// TwinCAT 3 PLC project PLC1
// ProgramVersion: 3.1.4020.4
// libraries:
//   Tc2_Standard, * (Beckhoff Automation GmbH)
//   Tc2_System, * (Beckhoff Automation GmbH)
//   Tc2_TcpIp, * (Beckhoff Automation GmbH)
//   Tc2_Utilities, * (Beckhoff Automation GmbH)
//   Tc3_Module, * (Beckhoff Automation GmbH)
// project tree:
//   HTTP/DUTs/ E_HTTP_Request_Type.TcDUT, ST_HTTP_Connection_Parameters.TcDUT, ST_HTTP_Parameter.TcDUT, ST_HTTP_Request.TcDUT, ST_HTTP_Response.TcDUT
//   HTTP/ FB_Http_Client.TcPOU
//   HTTP/GVLs/ GVL_HTTP.TcGVL
//   HTTP/Helper POUs/ FB_BinaryWriter.TcPOU, FB_GetHttpConnectionParams.TcPOU, F_BuildHttpGetRequest.TcPOU, F_BuildHttpPostRequest.TcPOU, F_MultiConcat12.TcPOU, F_MultiConcat6.TcPOU, F_ParseHttpResponse.TcPOU, F_ParseHttpUrl.TcPOU
//   HTTP/InfluxDb/ FB_Http_Client_Influx.TcPOU, F_BuildHttpPostRequest_InfluxDb.TcPOU
//   / PlcTask.TcTTO
//   POUs/ MAIN.TcPOU
// real-time tasks:
//   TASK PlcTask: cycle T#10ms, priority 20, ADS port 350

CONFIGURATION PLC1
    RESOURCE PLC ON TwinCAT3
        TASK PlcTask(INTERVAL := T#10ms, PRIORITY := 20);
        PROGRAM MAIN WITH PlcTask : MAIN;
    END_RESOURCE
END_CONFIGURATION

// ---- HTTP/DUTs/E_HTTP_Request_Type.TcDUT
TYPE E_HTTP_Request_Type :
(
	E_HTTP_Request_Type_GET := 0,
	E_HTTP_Request_Type_POST := 1
);
END_TYPE

// ---- HTTP/DUTs/ST_HTTP_Connection_Parameters.TcDUT
TYPE ST_HTTP_Connection_Parameters :
STRUCT
	bIsValid		: BOOL;
	sIpv4Address	: STRING;
	udPort			: UDINT;
	sHostName		: STRING;
	sRequestURI 	: STRING;
END_STRUCT
END_TYPE

// ---- HTTP/DUTs/ST_HTTP_Parameter.TcDUT
TYPE ST_HTTP_Parameter :
STRUCT
	sName	: STRING;
	sValue	: STRING;
END_STRUCT
END_TYPE

// ---- HTTP/DUTs/ST_HTTP_Request.TcDUT
TYPE ST_HTTP_Request :
STRUCT
	eHttpRequestType	: E_HTTP_Request_Type;
	arrParameters 		: ARRAY [0..HTTP_PARAMETERS_ARRAY_SIZE] OF ST_HTTP_Parameter;
END_STRUCT
END_TYPE

// ---- HTTP/DUTs/ST_HTTP_Response.TcDUT
TYPE ST_HTTP_Response :
STRUCT
	arrHeaders	: ARRAY [0..HTTP_RESPONSE_HEADER_ARRAY_SIZE] OF STRING;
	sContent	: STRING(255);
END_STRUCT
END_TYPE

// ---- HTTP/GVLs/GVL_HTTP.TcGVL
VAR_GLOBAL CONSTANT
	HTTP_SEND_DATA_ARRAY_SIZE 		: UDINT := 49999; 
	HTTP_RECEIVE_DATA_ARRAY_SIZE 	: UDINT := 9999; 
	HTTP_PARAMETERS_ARRAY_SIZE		: UDINT := 499;
	HTTP_RESPONSE_HEADER_ARRAY_SIZE	: UDINT := 20; 
END_VAR

// ---- POUs/MAIN.TcPOU
PROGRAM MAIN
VAR
	fbHttp_ClientPost	: FB_Http_Client;
	stHttpReqPost		: ST_HTTP_Request; 
	stHttpResponsePost	: ST_HTTP_Response;
	sResponsePost		: STRING(255);
	T1_TON				: TON;
	
	fbHttp_ClientGet	: FB_Http_Client;
	stHttpReqGet		: ST_HTTP_Request; 
	stHttpResponseGet	: ST_HTTP_Response;
	T2_TON				: TON;
	sResponseGet		: STRING(255);
	udCounter			: UDINT;
END_VAR

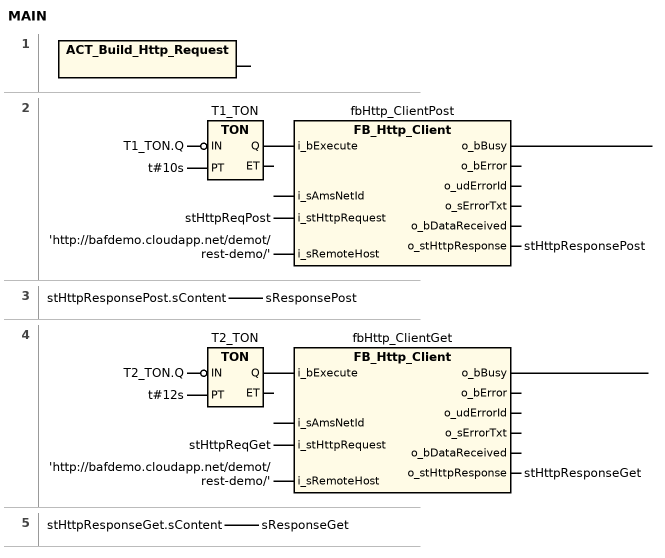
// NETWORK 1
ACT_Build_Http_Request();

// NETWORK 2
T1_TON(IN := NOT T1_TON.Q, PT := t#10s); // TON
fbHttp_ClientPost(
    i_bExecute := T1_TON.Q,
    i_stHttpRequest := stHttpReqPost,
    i_sRemoteHost := 'http://bafdemo.cloudapp.net/demot/rest-demo/',
    o_stHttpResponse => stHttpResponsePost); // FB_Http_Client

// NETWORK 3
sResponsePost := stHttpResponsePost.sContent;

// NETWORK 4
T2_TON(IN := NOT T2_TON.Q, PT := t#12s); // TON
fbHttp_ClientGet(
    i_bExecute := T2_TON.Q,
    i_stHttpRequest := stHttpReqGet,
    i_sRemoteHost := 'http://bafdemo.cloudapp.net/demot/rest-demo/',
    o_stHttpResponse => stHttpResponseGet); // FB_Http_Client

// NETWORK 5
sResponseGet := stHttpResponseGet.sContent;

ACTION ACT_Build_Http_Request:

(****  HTTP POST Example ********************************************************************************)

stHttpReqPost.eHttpRequestType 			:= E_HTTP_Request_Type.E_HTTP_Request_Type_POST;

stHttpReqPost.arrParameters[0].sName	:= 'passwd';
stHttpReqPost.arrParameters[0].sValue	:= 'TwoCats';

stHttpReqPost.arrParameters[1].sName	:= 'counter';
stHttpReqPost.arrParameters[1].sValue	:= UDINT_TO_STRING(udCounter);  udCounter := udCounter + 1;

stHttpReqPost.arrParameters[2].sName	:= 'cyclecount';
stHttpReqPost.arrParameters[2].sValue	:= UDINT_TO_STRING(_TaskInfo[1].CycleCount);

(*******************************************************************************************************)

(****  HTTP GET Example ********************************************************************************)

stHttpReqGet.eHttpRequestType 			:= E_HTTP_Request_Type.E_HTTP_Request_Type_GET;

stHttpReqGet.arrParameters[0].sName		:= 'passwd';
stHttpReqGet.arrParameters[0].sValue	:= 'TwoCats';

stHttpReqGet.arrParameters[1].sName		:= 'parameters';
stHttpReqGet.arrParameters[1].sValue	:= '1';

(*******************************************************************************************************)
END_ACTION

END_PROGRAM

// ---- HTTP/FB_Http_Client.TcPOU
FUNCTION_BLOCK FB_Http_Client
VAR_INPUT
	i_bExecute 			: BOOL;
	i_sAmsNetId			: STRING;
	i_stHttpRequest 	: ST_HTTP_Request;
	i_sRemoteHost		: STRING(255);
END_VAR
VAR_OUTPUT	
	o_bBusy				: BOOL;
	o_bError			: BOOL;
	o_udErrorId			: UDINT;
	o_sErrorTxt			: STRING;
	o_bDataReceived		: BOOL;	
	o_stHttpResponse	: ST_HTTP_Response;
END_VAR
VAR
	fbGetHttpConnectionParams: FB_GetHttpConnectionParams;
	fbSocketConnect		: FB_SocketConnect;
	fbSocketSend		: FB_SocketSend;
	fbSocketReceive		: FB_SocketReceive;
	fbSocketClose		: FB_SocketClose;
	bGetHttpConnectionParams: BOOL;
	bSocketConnect		: BOOL;
	bSocketSend			: BOOL;
	bSocketReceive		: BOOL;
	bSocketClose		: BOOL;
	nState				: INT := 10;
	hSocket				: T_HSOCKET;
	udBytesToSend		: UDINT;
	arrBytesToSend		: ARRAY[0..HTTP_SEND_DATA_ARRAY_SIZE] OF BYTE;
	tTimeOut			: TIME := T#10S;
	arrReceivedBytes	: ARRAY[0..HTTP_RECEIVE_DATA_ARRAY_SIZE] OF BYTE;
	bHttpConnParamsParamsParsed : BOOL;
	stHttpConnectionParams : ST_HTTP_Connection_Parameters;
	udReceivedBytes		: UDINT;
	Delay_TON			: TON;
END_VAR



CASE nState OF

10: (* Initial state *)
	nState := 20;
	
20:	(* Waiting for start *)

	IF i_bExecute THEN
		
		MEMSET(ADR(arrReceivedBytes), 0, SIZEOF(arrReceivedBytes));
		o_bDataReceived := FALSE;
		udReceivedBytes := 0;
		o_udErrorId		:= 0;
		o_bError 		:= FALSE;
		o_sErrorTxt 	:= '';
		o_bBusy 		:= TRUE;
		
		IF NOT bHttpConnParamsParamsParsed THEN
			bGetHttpConnectionParams := TRUE;
			nState := 25;
		ELSE
			bSocketConnect 	:= TRUE;
			nState 			:= 30;
		END_IF
		
	END_IF

25:	(* Waiting for addr resolved *)


	IF fbGetHttpConnectionParams.o_bError THEN
		o_udErrorId := fbGetHttpConnectionParams.o_nErrId;
		o_sErrorTxt := 'FB_GetHttpConnectionParams error';
		nState 		:= 100; 
	ELSIF fbGetHttpConnectionParams.o_bReady THEN
		stHttpConnectionParams := fbGetHttpConnectionParams.o_stHttpConnectionParams;
		bHttpConnParamsParamsParsed := TRUE;
		bSocketConnect 	:= TRUE;
		nState 			:= 30;
	END_IF	

30:	(* Waiting for connect *)

	IF fbSocketConnect.bError THEN
		o_udErrorId := fbSocketConnect.nErrId;
		o_sErrorTxt := 'FB_SocketConnect error';
		nState 		:= 100; 
	ELSIF NOT fbSocketConnect.bBusy THEN
		
		CASE i_stHttpRequest.eHttpRequestType OF 
			
			E_HTTP_Request_Type_GET:			
					udBytesToSend 	:= F_BuildHttpGetRequest(ADR(i_stHttpRequest), stHttpConnectionParams, arrBytesToSend);
							
			E_HTTP_Request_Type_POST:			
					udBytesToSend 	:= F_BuildHttpPostRequest(ADR(i_stHttpRequest), stHttpConnectionParams, arrBytesToSend);
							
		END_CASE

		bSocketSend		:= TRUE;
		nState 			:= 40; 		
	END_IF

40:	(* Waiting for send *) 

	IF fbSocketSend.bError THEN
		o_udErrorId := fbSocketSend.nErrId;
		o_sErrorTxt := 'FB_SocketSend error';
		nState 		:= 100; 
	ELSIF NOT fbSocketSend.bBusy THEN
		bSocketReceive	:= TRUE;
		nState 			:= 50; 		
	END_IF
	
50:	(* Waiting for receive *)

	// Timeout
	Delay_TON(IN := TRUE, PT := T#1500MS);
	
	IF fbSocketReceive.bError THEN
		Delay_TON(IN := FALSE);
		o_udErrorId := fbSocketReceive.nErrId;
		o_sErrorTxt := 'FB_SocketReceive error';
		nState 		:= 100; 
	ELSIF NOT fbSocketReceive.bBusy THEN
		IF fbSocketReceive.nRecBytes > 0 THEN
			Delay_TON(IN := FALSE);
			o_bDataReceived := TRUE;
			udReceivedBytes := fbSocketReceive.nRecBytes;
			o_stHttpResponse:= F_ParseHttpResponse(i_udNumOfBytes := udReceivedBytes, io_arrReceivedBytes:= arrReceivedBytes);
			bSocketClose	:= TRUE;
			nState 			:= 60;
		ELSIF Delay_TON.Q THEN
			Delay_TON(IN := FALSE);
			bSocketClose	:= TRUE;
			nState 			:= 60;
		ELSE
			bSocketReceive	:= TRUE;
		END_IF
	END_IF

60:	(* Waiting for close *)

	IF fbSocketClose.bError THEN
		o_udErrorId := fbSocketClose.nErrId;
		o_sErrorTxt := 'FB_SocketReceive error';
		nState 		:= 100; 
	ELSIF NOT fbSocketClose.bBusy THEN
		nState 	:= 10; 		
		o_bBusy := FALSE;
	END_IF

100:	(* Error *)

	o_bBusy  := FALSE;
	o_bError := TRUE;
	IF NOT i_bExecute THEN
		nState := 10;
	END_IF

END_CASE

ACT_FB_Calls();

bGetHttpConnectionParams := FALSE;
bSocketConnect 	:= FALSE;
bSocketSend 	:= FALSE;
bSocketReceive 	:= FALSE;
bSocketClose 	:= FALSE;

ACTION ACT_FB_Calls:
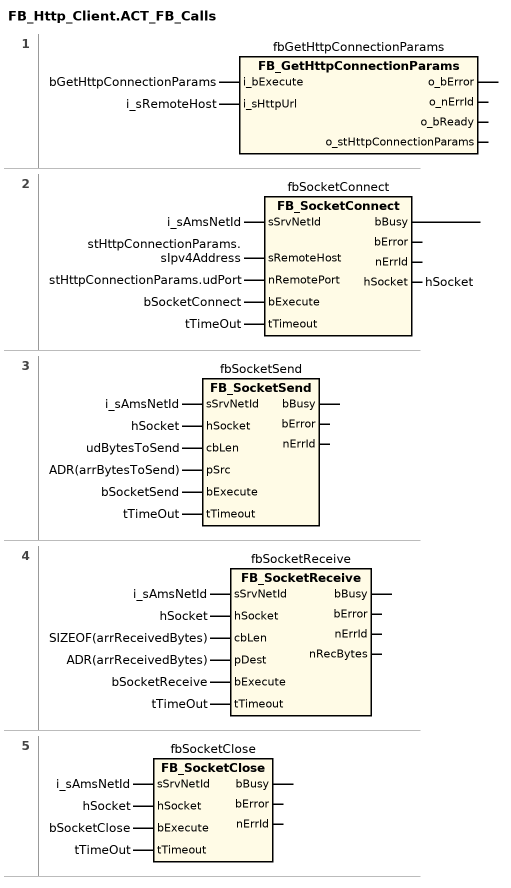
// NETWORK 1
fbGetHttpConnectionParams(i_bExecute := bGetHttpConnectionParams, i_sHttpUrl := i_sRemoteHost); // FB_GetHttpConnectionParams

// NETWORK 2
fbSocketConnect(
    sSrvNetId := i_sAmsNetId,
    sRemoteHost := stHttpConnectionParams.sIpv4Address,
    nRemotePort := stHttpConnectionParams.udPort,
    bExecute := bSocketConnect,
    tTimeout := tTimeOut,
    hSocket => hSocket); // FB_SocketConnect

// NETWORK 3
fbSocketSend(
    sSrvNetId := i_sAmsNetId,
    hSocket := hSocket,
    cbLen := udBytesToSend,
    pSrc := ADR(arrBytesToSend),
    bExecute := bSocketSend,
    tTimeout := tTimeOut); // FB_SocketSend

// NETWORK 4
fbSocketReceive(
    sSrvNetId := i_sAmsNetId,
    hSocket := hSocket,
    cbLen := SIZEOF(arrReceivedBytes),
    pDest := ADR(arrReceivedBytes),
    bExecute := bSocketReceive,
    tTimeout := tTimeOut); // FB_SocketReceive

// NETWORK 5
fbSocketClose(sSrvNetId := i_sAmsNetId, hSocket := hSocket, bExecute := bSocketClose, tTimeout := tTimeOut); // FB_SocketClose
END_ACTION

END_FUNCTION_BLOCK

// ---- HTTP/Helper POUs/FB_GetHttpConnectionParams.TcPOU
FUNCTION_BLOCK FB_GetHttpConnectionParams
VAR_INPUT
	i_bExecute	: BOOL;
	i_sHttpUrl	: T_MaxString;
END_VAR
VAR_OUTPUT
	o_bError	: BOOL;
	o_nErrId	: UDINT;
	o_bReady	: BOOL;
	o_stHttpConnectionParams : ST_HTTP_Connection_Parameters;
END_VAR
VAR
	fbGetHostAddrByName		: FB_GetHostAddrByName;
	stHttpConnectionParams 	: ST_HTTP_Connection_Parameters;
	execute_R_TRIG			: R_TRIG;
	getHostAddrBusy_F_TRIG	: F_TRIG;
	bExecute				: BOOL;
	bUrlValid: BOOL;
	nState: INT := 10;
END_VAR



CASE nState OF
	
10: (* init *)
	nState := 20;
	
20:	(* Waiting for start *)
	
	IF i_bExecute THEN
		(* Reset *)
		o_bReady := FALSE;
		o_bError := FALSE;
		o_nErrId := 0;
		MEMSET(ADR(o_stHttpConnectionParams), 0, SIZEOF(o_stHttpConnectionParams));
		
		IF F_ParseHttpUrl(i_sHttpUrl, stHttpConnectionParams) THEN
			IF stHttpConnectionParams.sHostName <> 'localhost' THEN

				nState := 30;
			ELSE
				stHttpConnectionParams.sIpv4Address := '127.0.0.1';	
				o_stHttpConnectionParams := stHttpConnectionParams;
				o_bReady := TRUE;
				nState := 20;			
			END_IF
		ELSE 
			o_bError := TRUE;
		END_IF
	END_IF

30:	(* Waiting for ready *)

	fbGetHostAddrByName(
		sHostName	:= stHttpConnectionParams.sHostName,
		bExecute 	:= TRUE,
		tTimeout 	:= T#10S
	);
	
	IF fbGetHostAddrByName.bError THEN
		fbGetHostAddrByName(bExecute := FALSE);
		o_bError := TRUE;
		o_nErrId := fbGetHostAddrByName.nErrID;
		nState := 100;
	ELSIF NOT fbGetHostAddrByName.bBusy THEN
		fbGetHostAddrByName(bExecute := FALSE);
		stHttpConnectionParams.sIpv4Address := fbGetHostAddrByName.sAddr;
		o_stHttpConnectionParams := stHttpConnectionParams;
		o_bReady := TRUE;
		nState := 20;
	END_IF
	
100: (* Error state*)

	IF NOT i_bExecute THEN
		nState := 10;
	END_IF

END_CASE

END_FUNCTION_BLOCK

// ---- HTTP/Helper POUs/F_ParseHttpUrl.TcPOU
FUNCTION F_ParseHttpUrl : BOOL
VAR_INPUT
	i_sUrl :T_MaxString;
END_VAR
VAR_IN_OUT 
	io_stConnectionParameters : ST_HTTP_Connection_Parameters;
END_VAR
VAR
	sUrl : T_MaxString;
	stConnectionParameters : ST_HTTP_Connection_Parameters;
	nPos: INT;
	nPosPort: INT;
END_VAR

sUrl := i_sUrl;

//the shortest form http://a.fi ==> 11 characters
IF LEN(sUrl) < 11 THEN
	F_ParseHttpUrl := FALSE;
	RETURN;
END_IF

// Parse the protocol
IF LEFT(sUrl, 5) = 'https' THEN
	// HTTPS is not supported
	F_ParseHttpUrl := FALSE;
	RETURN;
ELSIF LEFT(sUrl, 4) = 'http' THEN
	stConnectionParameters.udPort := 80;
	sUrl := RIGHT(sUrl, LEN(sUrl) - 4);
ELSE
	F_ParseHttpUrl := FALSE;
	RETURN;
END_IF

//Remove '://'
IF LEFT(sUrl, 3) = '://' THEN
	sUrl := RIGHT(sUrl, LEN(sUrl) - 3);
	// There is only domain + request uri left, minimun 4 characters (a.fi)
	IF LEN(sUrl) < 4 THEN 
		F_ParseHttpUrl := FALSE;
		RETURN;
	END_IF
ELSE
	F_ParseHttpUrl := FALSE;
	RETURN;
END_IF

// We have domain [+ port [+ request uri]] left
nPos := FIND(sUrl, '/');
nPosPort := FIND(sUrl, ':');

IF nPos = 0 THEN
	IF nPosPort > 0 THEN
		stConnectionParameters.sHostName := LEFT(sUrl, nPosPort-1);
		sUrl := RIGHT(sUrl, LEN(sUrl) - nPosPort);		
	ELSE
		stConnectionParameters.sHostName := sUrl;
	END_IF
	stConnectionParameters.sRequestURI := '/';
	io_stConnectionParameters := stConnectionParameters;
	F_ParseHttpUrl := TRUE;
ELSE
	IF nPosPort > 0 THEN
		stConnectionParameters.sHostName := LEFT(sUrl, nPosPort-1);
		sUrl := RIGHT(sUrl, LEN(sUrl) - nPosPort);		
		nPos := FIND(sUrl, '/');
		stConnectionParameters.udPort := STRING_TO_UDINT(LEFT(sUrl, nPos-1));
		sUrl := RIGHT(sUrl, LEN(sUrl) - nPos + 1);	
	ELSE
		stConnectionParameters.sHostName := LEFT(sUrl, nPos-1);
		sUrl := RIGHT(sUrl, LEN(sUrl) - nPos+1);
	END_IF	
	stConnectionParameters.sRequestURI := sUrl;
	io_stConnectionParameters := stConnectionParameters;
	F_ParseHttpUrl := TRUE;
END_IF

END_FUNCTION

// ---- HTTP/Helper POUs/F_BuildHttpGetRequest.TcPOU
FUNCTION F_BuildHttpGetRequest : UDINT
VAR_INPUT
	i_pHttpRequest 		: POINTER TO ST_HTTP_Request;
	i_stHttpConnParams	: ST_HTTP_Connection_Parameters;
END_VAR
VAR_IN_OUT
	io_arrBytesToSend	: ARRAY[0..HTTP_SEND_DATA_ARRAY_SIZE] OF BYTE;
END_VAR
VAR
	sData				: T_MaxString;
	i					: INT;
	nContentLength		: DINT;
	fbBinaryWriter		: FB_BinaryWriter;
	sRequestString		: STRING(255);
END_VAR


fbBinaryWriter.Init(ADR(io_arrBytesToSend), SIZEOF(io_arrBytesToSend));
MEMSET(ADR(io_arrBytesToSend), 0, SIZEOF(io_arrBytesToSend));

fbBinaryWriter.WriteString('GET ');
fbBinaryWriter.WriteString(i_stHttpConnParams.sRequestURI);

// Write the GET request into request uri
FOR i := 0 TO UDINT_TO_INT(HTTP_PARAMETERS_ARRAY_SIZE) DO 
	IF LEN(i_pHttpRequest^.arrParameters[i].sName) > 0 THEN
		IF i = 0 THEN fbBinaryWriter.WriteString('?'); END_IF
		IF i > 0 THEN fbBinaryWriter.WriteString('&'); END_IF
		fbBinaryWriter.WriteString(i_pHttpRequest^.arrParameters[i].sName);
		fbBinaryWriter.WriteString('=');
		fbBinaryWriter.WriteString(i_pHttpRequest^.arrParameters[i].sValue);
	END_IF
END_FOR

fbBinaryWriter.WriteString(' HTTP/1.0$R$N'); // Lets use HTTP 1.0 because responce with "Transfer-Encoding:chunked is much more complex to parse
fbBinaryWriter.WriteString('Host: ');
fbBinaryWriter.WriteString(i_stHttpConnParams.sHostName);
fbBinaryWriter.WriteString(' $R$N');
fbBinaryWriter.WriteString('User-Agent: TwinCAT HttpClient$R$N');

// Calculate the length of data
FOR i := 0 TO UDINT_TO_INT(HTTP_PARAMETERS_ARRAY_SIZE) DO 
	IF LEN(i_pHttpRequest^.arrParameters[i].sName) > 0 THEN
		IF i > 0 THEN nContentLength := nContentLength + 1; END_IF
		nContentLength := nContentLength + LEN(i_pHttpRequest^.arrParameters[i].sName) + LEN(i_pHttpRequest^.arrParameters[i].sValue) + 1;
	END_IF
END_FOR	
fbBinaryWriter.WriteString('$R$N$R$N');
	
sRequestString := fbBinaryWriter.ToString;

F_BuildHttpGetRequest := fbBinaryWriter.Length;

(****** GET Request principle ***********************************************************************

fbBinaryWriter.WriteString('GET /demot/rest-demo/?'param1=1&param2=2&param3=3' HTTP/1.1$R$N');
fbBinaryWriter.WriteString('Host: bafdemo.cloudapp.net $R$N');
fbBinaryWriter.WriteString('User-Agent: TwinCAT 3.1$R$N');
fbBinaryWriter.WriteString('$R$N$R$N');

***************************************************************************************************)

END_FUNCTION

// ---- HTTP/Helper POUs/FB_BinaryWriter.TcPOU
FUNCTION_BLOCK FB_BinaryWriter
VAR_INPUT
	i_pDestAddr		: POINTER TO BYTE;
	i_udDestAddrLen	: UDINT;
END_VAR
VAR_OUTPUT
END_VAR
VAR
	pDestAddr		: POINTER TO BYTE;
	udDestAddrLen	: UDINT;
	udCurrentLen 	: UDINT;
END_VAR

METHOD Init : BOOL
VAR_INPUT
	i_pDestAddr		: POINTER TO BYTE;
	i_udDestAddrLen	: UDINT;
END_VAR
pDestAddr 		:= i_pDestAddr;
udDestAddrLen 	:=i_udDestAddrLen;
udCurrentLen 	:= 0;

(* Reset the stream *)
MEMSET(i_pDestAddr, 0, i_udDestAddrLen);
END_METHOD

PROPERTY Length : udint
GET
Length := udCurrentLen;
END_GET
END_PROPERTY

METHOD SetPosition : BOOL
VAR_INPUT
	i_udPosition : UDINT;
END_VAR
IF i_udPosition <= udDestAddrLen THEN
	udCurrentLen := i_udPosition;
	SetPosition := TRUE;
ELSE
	SetPosition := FALSE;
END_IF
END_METHOD

PROPERTY ToString : STRING(255)
GET
VAR
	s255String : STRING(255);
	length : UDINT;
END_VAR
s255String := '';
length := MIN(udCurrentLen, DINT_TO_UDINT(SIZEOF(s255String)));
MEMCPY(ADR(s255String), pDestAddr, length);
ToString := s255String;
END_GET
END_PROPERTY

METHOD WriteString : BOOL
VAR_INPUT
	i_sStringToAppend : T_MaxString;
END_VAR
VAR
	udStringLen: UDINT;
END_VAR

udStringLen := DINT_TO_UDINT(LEN(i_sStringToAppend));

(* Only write if there's memory free for writing *)
IF udCurrentLen + udStringLen < udDestAddrLen THEN
	MEMCPY(pDestAddr + udCurrentLen, ADR(i_sStringToAppend), udStringLen);
	udCurrentLen := udCurrentLen + udStringLen;
	WriteString := TRUE;
ELSE
	WriteString := FALSE;
END_IF
END_METHOD

END_FUNCTION_BLOCK

// ---- HTTP/Helper POUs/F_BuildHttpPostRequest.TcPOU
FUNCTION F_BuildHttpPostRequest : UDINT
VAR_INPUT
	i_pHttpRequest 		: POINTER TO ST_HTTP_Request;
	i_stHttpConnParams	: ST_HTTP_Connection_Parameters;
END_VAR
VAR_IN_OUT
	io_arrBytesToSend	: ARRAY[0..HTTP_SEND_DATA_ARRAY_SIZE] OF BYTE;
END_VAR
VAR
	sData				: T_MaxString;
	i					: INT;
	nContentLength		: DINT;
	fbBinaryWriter		: FB_BinaryWriter;
	sRequestString		: STRING(255);
END_VAR


fbBinaryWriter.Init(ADR(io_arrBytesToSend), SIZEOF(io_arrBytesToSend));
MEMSET(ADR(io_arrBytesToSend), 0, SIZEOF(io_arrBytesToSend));

fbBinaryWriter.WriteString('POST ');
fbBinaryWriter.WriteString(i_stHttpConnParams.sRequestURI);
fbBinaryWriter.WriteString(' HTTP/1.0$R$N'); // Lets use HTTP 1.0 because responce with "Transfer-Encoding:chunked is much more complex to parse
fbBinaryWriter.WriteString('Host: ');
fbBinaryWriter.WriteString(i_stHttpConnParams.sHostName);
fbBinaryWriter.WriteString(' $R$N');
fbBinaryWriter.WriteString('User-Agent: TwinCAT HttpClient$R$N');
fbBinaryWriter.WriteString('Content-Type: application/x-www-form-urlencoded$R$N');

// Calculate the length of data
FOR i := 0 TO UDINT_TO_INT(HTTP_PARAMETERS_ARRAY_SIZE) DO 
	IF LEN(i_pHttpRequest^.arrParameters[i].sName) > 0 THEN
		IF i > 0 THEN nContentLength := nContentLength + 1; END_IF
		nContentLength := nContentLength + LEN(i_pHttpRequest^.arrParameters[i].sName) + LEN(i_pHttpRequest^.arrParameters[i].sValue) + 1;
	END_IF
END_FOR	

fbBinaryWriter.WriteString(CONCAT('Content-Length: ', DINT_TO_STRING(nContentLength)));


// Http request headers always end to double new line		
fbBinaryWriter.WriteString('$R$N$R$N');

// Write the POST data into request body
FOR i := 0 TO UDINT_TO_INT(HTTP_PARAMETERS_ARRAY_SIZE) DO 
	IF LEN(i_pHttpRequest^.arrParameters[i].sName) > 0 THEN
		IF i > 0 THEN fbBinaryWriter.WriteString('&'); END_IF
		fbBinaryWriter.WriteString(i_pHttpRequest^.arrParameters[i].sName);
		fbBinaryWriter.WriteString('=');
		fbBinaryWriter.WriteString(i_pHttpRequest^.arrParameters[i].sValue);
	END_IF
END_FOR

// Http request body always ends to new line		
fbBinaryWriter.WriteString('$R$N');


sRequestString := fbBinaryWriter.ToString;
F_BuildHttpPostRequest := fbBinaryWriter.Length;

(****** POST Request principle ***********************************************************************

sPostData = 'param1=1&param2=2&param3=3';
fbBinaryWriter.WriteString('POST /demot/rest-demo/ HTTP/1.1$R$N');
fbBinaryWriter.WriteString('Host: bafdemo.cloudapp.net $R$N');
fbBinaryWriter.WriteString('User-Agent: TwinCAT 3.1$R$N');
fbBinaryWriter.WriteString('Content-Type: application/x-www-form-urlencoded$R$N');
fbBinaryWriter.WriteString(CONCAT('Content-Length: ', DINT_TO_STRING(LEN(sPostData))));
fbBinaryWriter.WriteString('$R$N$R$N');
fbBinaryWriter.WriteString(sPostData);
fbBinaryWriter.WriteString('$R$N');

******************************************************************************************************)

END_FUNCTION

// ---- HTTP/Helper POUs/F_ParseHttpResponse.TcPOU
FUNCTION F_ParseHttpResponse : ST_HTTP_Response
VAR_INPUT
	i_udNumOfBytes 	: UDINT;
END_VAR
VAR_IN_OUT
	io_arrReceivedBytes	: ARRAY[0..HTTP_RECEIVE_DATA_ARRAY_SIZE] OF BYTE;
END_VAR
VAR
	i				: UDINT;
	headerIndex		: UDINT;
	stHttpResp 		: ST_HTTP_Response;
	pReceivedBytes	: POINTER TO BYTE;
	udNumOfBytes	: UDINT;
	udBytesToCopy	: UDINT;
	start: UDINT;
	arrDummyArray	: ARRAY [0..HTTP_RECEIVE_DATA_ARRAY_SIZE] OF BYTE;
	length: UDINT;
END_VAR


IF i_udNumOfBytes < 20 THEN
	RETURN;
END_IF

headerIndex 	:= 0;
udNumOfBytes := MIN(i_udNumOfBytes, HTTP_RECEIVE_DATA_ARRAY_SIZE);

FOR i := 0 TO udNumOfBytes - 3 DO
	
	IF io_arrReceivedBytes[i] = 13 AND io_arrReceivedBytes[i+1] = 10 AND io_arrReceivedBytes[i+2] = 13 AND io_arrReceivedBytes[i+3] = 10 THEN
		
		// We've found the double linefeed ($R$N$R$N) ==> the rest of messafe is the actual content we are interested
		
		length := i - start;
		MEMCPY(ADR(arrDummyArray), ADR(io_arrReceivedBytes[start]), length);
		arrDummyArray[length] := 0;
		MEMCPY(ADR(stHttpResp.arrHeaders[headerIndex]), ADR(arrDummyArray), length + 1);
		
		udBytesToCopy := MIN(udNumOfBytes - i + 3, SIZEOF(stHttpResp.sContent));
		MEMCPY(ADR(stHttpResp.sContent), ADR(io_arrReceivedBytes[i+4]), udBytesToCopy);
		
		EXIT;
		
	ELSIF io_arrReceivedBytes[i] = 13 AND io_arrReceivedBytes[i+1] = 10 THEN
		
		// We've found a single linefeed ($R$N) ==> a single response header ends here
		
		length := i - start;
		MEMCPY(ADR(arrDummyArray), ADR(io_arrReceivedBytes[start]), length);
		arrDummyArray[length] := 0;
		MEMCPY(ADR(stHttpResp.arrHeaders[headerIndex]), ADR(arrDummyArray), length + 1);
		start := i + 2;
		headerIndex := headerIndex + 1;
		
		IF headerIndex > HTTP_RESPONSE_HEADER_ARRAY_SIZE THEN
			EXIT;
		END_IF
		
	END_IF
END_FOR
F_ParseHttpResponse := stHttpResp;

END_FUNCTION

// ---- HTTP/Helper POUs/F_MultiConcat12.TcPOU
FUNCTION F_MultiConcat12 : STRING(255)
VAR_INPUT
	i_str1	: STRING;
	i_str2	: STRING;
	i_str3	: STRING;
	i_str4	: STRING;
	i_str5	: STRING;
	i_str6	: STRING;
	i_str7	: STRING;
	i_str8	: STRING;
	i_str9	: STRING;
	i_str10	: STRING;
	i_str11	: STRING;
	i_str12	: STRING;
END_VAR
VAR
	sText:	STRING(255);
END_VAR


sText := CONCAT(i_str1, i_str2);
sText := CONCAT(sText, i_str3);
sText := CONCAT(sText, i_str4);
sText := CONCAT(sText, i_str5);
sText := CONCAT(sText, i_str6);
sText := CONCAT(sText, i_str7);
sText := CONCAT(sText, i_str8);
sText := CONCAT(sText, i_str9);
sText := CONCAT(sText, i_str10);
sText := CONCAT(sText, i_str11);
sText := CONCAT(sText, i_str12);

F_MultiConcat12 := sText;

END_FUNCTION

// ---- HTTP/Helper POUs/F_MultiConcat6.TcPOU
FUNCTION F_MultiConcat6 : STRING(255)
VAR_INPUT
	i_str1	: STRING;
	i_str2	: STRING;
	i_str3	: STRING;
	i_str4	: STRING;
	i_str5	: STRING;
	i_str6	: STRING;
END_VAR
VAR
	sText:	STRING(255);
END_VAR


sText := CONCAT(i_str1, i_str2);
sText := CONCAT(sText, i_str3);
sText := CONCAT(sText, i_str4);
sText := CONCAT(sText, i_str5);
sText := CONCAT(sText, i_str6);

F_MultiConcat6 := sText;

END_FUNCTION

// ---- HTTP/InfluxDb/FB_Http_Client_Influx.TcPOU
FUNCTION_BLOCK FB_Http_Client_Influx
VAR_INPUT
	i_bExecute 			: BOOL;
	i_sAmsNetId			: STRING;
	i_sRemoteHost		: STRING(255);
	i_nBytesToSend		: UDINT;
END_VAR
VAR_IN_OUT
	io_arrBytesToSend		: ARRAY[0..HTTP_SEND_DATA_ARRAY_SIZE] OF BYTE;
END_VAR
VAR_OUTPUT	
	o_bBusy				: BOOL;
	o_bError			: BOOL;
	o_udErrorId			: UDINT;
	o_sErrorTxt			: STRING;
	o_bDataReceived		: BOOL;	
	o_stHttpResponse	: ST_HTTP_Response;
END_VAR
VAR
	fbGetHttpConnectionParams: FB_GetHttpConnectionParams;
	fbSocketConnect		: FB_SocketConnect;
	fbSocketSend		: FB_SocketSend;
	fbSocketReceive		: FB_SocketReceive;
	fbSocketClose		: FB_SocketClose;
	bGetHttpConnectionParams: BOOL;
	bSocketConnect		: BOOL;
	bSocketSend			: BOOL;
	bSocketReceive		: BOOL;
	bSocketClose		: BOOL;
	nState				: INT := 10;
	hSocket				: T_HSOCKET;
	udBytesToSend		: UDINT;
	arrBytesToSend		: ARRAY[0..HTTP_SEND_DATA_ARRAY_SIZE] OF BYTE;
	udReceivedBytes		: UDINT;
	arrReceivedBytes	: ARRAY[0..HTTP_RECEIVE_DATA_ARRAY_SIZE] OF BYTE;
	tTimeOut			: TIME := T#10S;
	bHttpConnParamsParamsParsed : BOOL;
	stHttpConnectionParams : ST_HTTP_Connection_Parameters;
	Delay_TON: TON;
END_VAR



CASE nState OF

10: (* Initial state *)
	nState := 20;
	
20:	(* Waiting for start *)

	IF i_bExecute THEN
		
		MEMSET(ADR(arrReceivedBytes), 0, SIZEOF(arrReceivedBytes));
		o_bDataReceived := FALSE;
		udReceivedBytes := 0;
		o_udErrorId		:= 0;
		o_bError 		:= FALSE;
		o_sErrorTxt 	:= '';
		o_bBusy 		:= TRUE;
		
		IF NOT bHttpConnParamsParamsParsed THEN
			bGetHttpConnectionParams := TRUE;
			nState := 25;
		ELSE
			bSocketConnect 	:= TRUE;
			nState 			:= 30;
		END_IF
		
	END_IF

25:	(* Waiting for addr resolved *)


	IF fbGetHttpConnectionParams.o_bError THEN
		o_udErrorId := fbGetHttpConnectionParams.o_nErrId;
		o_sErrorTxt := 'FB_GetHttpConnectionParams error';
		nState 		:= 100; 
	ELSIF fbGetHttpConnectionParams.o_bReady THEN
		stHttpConnectionParams := fbGetHttpConnectionParams.o_stHttpConnectionParams;
		bHttpConnParamsParamsParsed := TRUE;
		bSocketConnect 	:= TRUE;
		nState 			:= 30;
	END_IF	

30:	(* Waiting for connect *)

	IF fbSocketConnect.bError THEN
		o_udErrorId := fbSocketConnect.nErrId;
		o_sErrorTxt := 'FB_SocketConnect error';
		nState 		:= 100; 
	ELSIF NOT fbSocketConnect.bBusy THEN
		
		udBytesToSend 	:= F_BuildHttpPostRequest_InfluxDb(stHttpConnectionParams, i_nBytesToSend, io_arrBytesToSend, arrBytesToSend);
		bSocketSend		:= TRUE;
		nState 			:= 40;
 		
	END_IF

40:	(* Waiting for send *) 

	IF fbSocketSend.bError THEN
		o_udErrorId := fbSocketSend.nErrId;
		o_sErrorTxt := 'FB_SocketSend error';
		nState 		:= 100; 
	ELSIF NOT fbSocketSend.bBusy THEN
		bSocketReceive	:= TRUE;
		nState 			:= 50; 		
	END_IF
	
50:	(* Waiting for receive *)

	// Timeout
	Delay_TON(IN := TRUE, PT := T#1500MS);
	
	IF fbSocketReceive.bError THEN
		Delay_TON(IN := FALSE);
		o_udErrorId := fbSocketReceive.nErrId;
		o_sErrorTxt := 'FB_SocketReceive error';
		nState 		:= 100; 
	ELSIF NOT fbSocketReceive.bBusy THEN
		IF fbSocketReceive.nRecBytes > 0 THEN
			Delay_TON(IN := FALSE);
			o_bDataReceived := TRUE;
			udReceivedBytes := fbSocketReceive.nRecBytes;
			o_stHttpResponse:= F_ParseHttpResponse(i_udNumOfBytes := udReceivedBytes, io_arrReceivedBytes:= arrReceivedBytes);
			bSocketClose	:= TRUE;
			nState 			:= 60;
		ELSIF Delay_TON.Q THEN
			Delay_TON(IN := FALSE);
			bSocketClose	:= TRUE;
			nState 			:= 60;
		ELSE
			bSocketReceive	:= TRUE;
		END_IF
	END_IF

60:	(* Waiting for close *)

	IF fbSocketClose.bError THEN
		o_udErrorId := fbSocketClose.nErrId;
		o_sErrorTxt := 'FB_SocketReceive error';
		nState 		:= 100; 
	ELSIF NOT fbSocketClose.bBusy THEN
		nState 	:= 10; 		
		o_bBusy := FALSE;
	END_IF

100:	(* Error *)

	o_bBusy  := FALSE;
	o_bError := TRUE;
	IF NOT i_bExecute THEN
		nState := 10;
	END_IF

END_CASE

ACT_FB_Calls();

bGetHttpConnectionParams := FALSE;
bSocketConnect 	:= FALSE;
bSocketSend 	:= FALSE;
bSocketReceive 	:= FALSE;
bSocketClose 	:= FALSE;

ACTION ACT_FB_Calls:
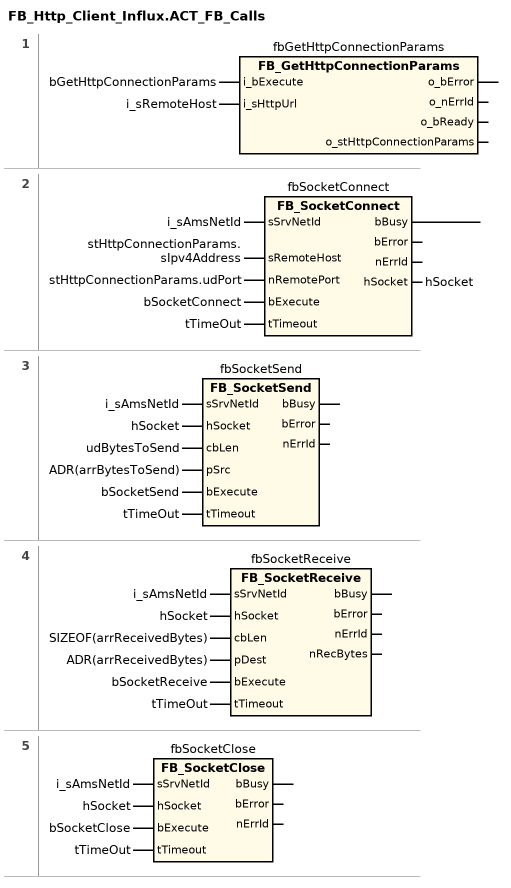
// NETWORK 1
fbGetHttpConnectionParams(i_bExecute := bGetHttpConnectionParams, i_sHttpUrl := i_sRemoteHost); // FB_GetHttpConnectionParams

// NETWORK 2
fbSocketConnect(
    sSrvNetId := i_sAmsNetId,
    sRemoteHost := stHttpConnectionParams.sIpv4Address,
    nRemotePort := stHttpConnectionParams.udPort,
    bExecute := bSocketConnect,
    tTimeout := tTimeOut,
    hSocket => hSocket); // FB_SocketConnect

// NETWORK 3
fbSocketSend(
    sSrvNetId := i_sAmsNetId,
    hSocket := hSocket,
    cbLen := udBytesToSend,
    pSrc := ADR(arrBytesToSend),
    bExecute := bSocketSend,
    tTimeout := tTimeOut); // FB_SocketSend

// NETWORK 4
fbSocketReceive(
    sSrvNetId := i_sAmsNetId,
    hSocket := hSocket,
    cbLen := SIZEOF(arrReceivedBytes),
    pDest := ADR(arrReceivedBytes),
    bExecute := bSocketReceive,
    tTimeout := tTimeOut); // FB_SocketReceive

// NETWORK 5
fbSocketClose(sSrvNetId := i_sAmsNetId, hSocket := hSocket, bExecute := bSocketClose, tTimeout := tTimeOut); // FB_SocketClose
END_ACTION

END_FUNCTION_BLOCK

// ---- HTTP/InfluxDb/F_BuildHttpPostRequest_InfluxDb.TcPOU
FUNCTION F_BuildHttpPostRequest_InfluxDb : UDINT
VAR_INPUT
	i_stHttpConnParams	: ST_HTTP_Connection_Parameters;
	i_nBytesToSend 		: UDINT;
END_VAR
VAR_IN_OUT
	io_arrInFluxData	: ARRAY[0..HTTP_SEND_DATA_ARRAY_SIZE] OF BYTE;
	io_arrBytesToSend	: ARRAY[0..HTTP_SEND_DATA_ARRAY_SIZE] OF BYTE;
END_VAR
VAR
	sData				: T_MaxString;
	i					: INT;
	nContentLength		: DINT;
	fbBinaryWriter		: FB_BinaryWriter;
	sRequestString		: STRING(255);
END_VAR


fbBinaryWriter.Init(ADR(io_arrBytesToSend), SIZEOF(io_arrBytesToSend));
MEMSET(ADR(io_arrBytesToSend), 0, SIZEOF(io_arrBytesToSend));

fbBinaryWriter.WriteString('POST ');
fbBinaryWriter.WriteString(i_stHttpConnParams.sRequestURI);
fbBinaryWriter.WriteString(' HTTP/1.1$R$N');
fbBinaryWriter.WriteString('Host: ');
fbBinaryWriter.WriteString(i_stHttpConnParams.sHostName);
fbBinaryWriter.WriteString(' $R$N');
fbBinaryWriter.WriteString('User-Agent: TwinCAT HttpClient$R$N');
fbBinaryWriter.WriteString('Content-Type: application/x-www-form-urlencoded$R$N');

// Calculate the length of data
fbBinaryWriter.WriteString(CONCAT('Content-Length: ', UDINT_TO_STRING(i_nBytesToSend)));

// Http request headers always end to double new line		
fbBinaryWriter.WriteString('$R$N$R$N');
// Copy the influx data into http request 
MEMCPY(ADR(io_arrBytesToSend[fbBinaryWriter.Length]), ADR(io_arrInFluxData), i_nBytesToSend);
fbBinaryWriter.SetPosition(fbBinaryWriter.Length + i_nBytesToSend);
// Http request body always ends to new line		
fbBinaryWriter.WriteString('$R$N');


sRequestString := fbBinaryWriter.ToString;
F_BuildHttpPostRequest_InfluxDb := fbBinaryWriter.Length;

(****** POST Request principle ***********************************************************************

sPostData = 'param1=1&param2=2&param3=3';
fbBinaryWriter.WriteString('POST /demot/rest-demo/ HTTP/1.1$R$N');
fbBinaryWriter.WriteString('Host: bafdemo.cloudapp.net $R$N');
fbBinaryWriter.WriteString('User-Agent: TwinCAT 3.1$R$N');
fbBinaryWriter.WriteString('Content-Type: application/x-www-form-urlencoded$R$N');
fbBinaryWriter.WriteString(CONCAT('Content-Length: ', DINT_TO_STRING(LEN(sPostData))));
fbBinaryWriter.WriteString('$R$N$R$N');
fbBinaryWriter.WriteString(sPostData);
fbBinaryWriter.WriteString('$R$N');

******************************************************************************************************)

END_FUNCTION
